// TwinCAT 3 PLC project IvS_Alpaca
// ProgramVersion: 3.1.4024.0
// libraries:
//   Tc2_Standard, * (Beckhoff Automation GmbH)
//   Tc2_System, * (Beckhoff Automation GmbH)
//   Tc2_Utilities, * (Beckhoff Automation GmbH)
//   Tc3_IotBase, * (Beckhoff Automation GmbH)
//   Tc3_JsonXml, * (Beckhoff Automation GmbH)
//   Tc3_Module, * (Beckhoff Automation GmbH)
//   VisuDialogs, * (System)
// project tree:
//   DUTs/Alpaca/ E_AlpacaCoverState.TcDUT, E_AlpacaStatusCode.TcDUT, ST_AlpacaGetBool.TcDUT, ST_AlpacaGetCoverState.TcDUT, ST_AlpacaGetDint.TcDUT, ST_AlpacaGetLreal.TcDUT, ST_AlpacaGetRequest.TcDUT, ST_AlpacaPutMove.TcDUT, ST_AlpacaPutNoArgs.TcDUT, ST_AlpacaPutRequest.TcDUT, ST_AlpacaPutSlewToAltAz.TcDUT, ST_AlpacaPutSlewToCoordinates.TcDUT, ST_AlpacaPutTracking.TcDUT
//   DUTs/AsaTelescope/ E_AsaTelescopeRequests.TcDUT, ST_AsaTelescopeGetters.TcDUT, ST_AsaTelescopePutters.TcDUT
//   / GlobalTextList.TcGTLO, PlcTask.TcTTO, Visualization Manager.TcVMO (not stored)
//   POUs/Alpaca/ FB_AlpacaGet.TcPOU, FB_AlpacaPut.TcPOU, F_AlpacaFormatUri.TcPOU
//   POUs/AsaTelescope/ FB_AsaTelescope.TcPOU
//   POUs/ MAIN.TcPOU
//   VISUs/Alpaca/ VISU_AlpacaGetBool.TcVIS, VISU_AlpacaGetCoverState.TcVIS, VISU_AlpacaGetLreal.TcVIS, VISU_AlpacaPutMove.TcVIS, VISU_AlpacaPutNoArgs.TcVIS, VISU_AlpacaPutRequest.TcVIS, VISU_AlpacaPutSlewToAltAz.TcVIS, VISU_AlpacaPutSlewToCoordinates.TcVIS, VISU_AlpacaPutTracking.TcVIS
//   VISUs/AsaTelescope/ VISU_AsaTelescope.TcVIS
//   VISUs/ VISU_MAIN.TcVIS
// real-time tasks:
//   TASK PlcTask: cycle T#10ms, priority 20, ADS port 350

CONFIGURATION IvS_Alpaca
    RESOURCE PLC ON TwinCAT3
        TASK PlcTask(INTERVAL := T#10ms, PRIORITY := 20);
        PROGRAM MAIN WITH PlcTask : MAIN;
    END_RESOURCE
END_CONFIGURATION

// ---- DUTs/Alpaca/E_AlpacaCoverState.TcDUT
{attribute 'qualified_only'}
{attribute 'to_string'}
TYPE E_AlpacaCoverState :
(
	NOT_PRESENT := 0,
    CLOSED      := 1,
    MOVING      := 2,
    OPEN        := 3,
    UNKNOWN     := 4,
    ERROR       := 5
) DINT := UNKNOWN;
END_TYPE

// ---- DUTs/Alpaca/E_AlpacaStatusCode.TcDUT
{attribute 'qualified_only'}
{attribute 'strict'}
TYPE E_AlpacaStatusCode :
(
    NOTSET                          := 0,
	OK                              := 1,
    ERROR                           := 2,
    ERROR_WRONG_CONVERSION          := 3,
    ERROR_WRONG_RESPONSE_MEMBER     := 4,
    ERROR_WRONG_RESPONSE_CONTENT    := 5,
    ERROR_WRONG_HTTP_STATUS_CODE    := 6,
    ERROR_OTHER_COMMAND_SCHEDULED   := 7
);
END_TYPE

// ---- DUTs/Alpaca/ST_AlpacaGetBool.TcDUT
TYPE ST_AlpacaGetBool EXTENDS ST_AlpacaGetRequest:
STRUCT
    bValue : BOOL;
END_STRUCT
END_TYPE

// ---- DUTs/Alpaca/ST_AlpacaGetCoverState.TcDUT
TYPE ST_AlpacaGetCoverState EXTENDS ST_AlpacaGetDint :
STRUCT
    eValue : E_AlpacaCoverState;
    sValue : STRING;
END_STRUCT
END_TYPE

// ---- DUTs/Alpaca/ST_AlpacaGetDint.TcDUT
TYPE ST_AlpacaGetDint EXTENDS ST_AlpacaGetRequest:
STRUCT
    nValue : DINT;
END_STRUCT
END_TYPE

// ---- DUTs/Alpaca/ST_AlpacaGetLreal.TcDUT
TYPE ST_AlpacaGetLreal EXTENDS ST_AlpacaGetRequest:
STRUCT
    lrValue : LREAL;
END_STRUCT
END_TYPE

// ---- DUTs/Alpaca/ST_AlpacaGetRequest.TcDUT
// Common base class for the "Get" requests
TYPE ST_AlpacaGetRequest :
STRUCT
    sName       : STRING;
    eStatusCode : E_AlpacaStatusCode;
    rAge        : REAL;                 // age of the last reading, in seconds, since the last loop start
END_STRUCT
END_TYPE

// ---- DUTs/Alpaca/ST_AlpacaPutMove.TcDUT
TYPE ST_AlpacaPutMove EXTENDS ST_AlpacaPutRequest:
STRUCT
    // inputs
    i_Position : DINT;
END_STRUCT
END_TYPE

// ---- DUTs/Alpaca/ST_AlpacaPutNoArgs.TcDUT
TYPE ST_AlpacaPutNoArgs EXTENDS ST_AlpacaPutRequest:
STRUCT
    // just for the sake of semantics, our 'No args' structure extends
    // our common "put" request structure, but it doesn't add any members.
END_STRUCT
END_TYPE

// ---- DUTs/Alpaca/ST_AlpacaPutRequest.TcDUT
// Common base class for the "Put" requests
TYPE ST_AlpacaPutRequest :
STRUCT
    sName           : STRING;
    bExecute        : BOOL;
    eStatusCode     : E_AlpacaStatusCode;
    nErrorCode      : DINT;
    sErrorMessage   : STRING;
END_STRUCT
END_TYPE

// ---- DUTs/Alpaca/ST_AlpacaPutSlewToAltAz.TcDUT
TYPE ST_AlpacaPutSlewToAltAz EXTENDS ST_AlpacaPutRequest:
STRUCT
    // inputs
    i_lrAltitude    : LREAL;
    i_lrAzimuth     : LREAL;
END_STRUCT
END_TYPE

// ---- DUTs/Alpaca/ST_AlpacaPutSlewToCoordinates.TcDUT
TYPE ST_AlpacaPutSlewToCoordinates EXTENDS ST_AlpacaPutRequest:
STRUCT
    // inputs
    i_lrRightAscension  : LREAL;
    i_lrDeclination     : LREAL;
END_STRUCT
END_TYPE

// ---- DUTs/Alpaca/ST_AlpacaPutTracking.TcDUT
TYPE ST_AlpacaPutTracking EXTENDS ST_AlpacaPutRequest:
STRUCT
    // inputs
    i_bTracking : BOOL;
END_STRUCT
END_TYPE

// ---- DUTs/AsaTelescope/E_AsaTelescopeRequests.TcDUT
{attribute 'qualified_only'}
TYPE E_AsaTelescopeRequests :
(
    // the data below gets read continuously in order from top to bottom
    RIGHT_ASCENSION := 0,
    DECLINATION,
    AZIMUTH,
    ALTITUDE,
    SLEWING,
    TARGET_RIGHT_ASCENSION,
    TARGET_DECLINATION,
    M2_POSITION,
    COVER_STATE,
    
    // COMMANDS
    // ==================================================================
    // special state meaning no state requested
    NO_COMMAND,
    // add all commands below (order is not relevant)
    ABORT_SLEW,
    SLEW_TO_ALTAZ,
    SLEW_TO_COORDINATES,
    OPEN_COVER,
    CLOSE_COVER,
    TRACKING,
    M2_MOVE
);
END_TYPE

// ---- DUTs/AsaTelescope/ST_AsaTelescopeGetters.TcDUT
TYPE ST_AsaTelescopeGetters :
STRUCT
    stRightAscension          : ST_AlpacaGetLreal      := (sName := 'Right Ascension');
    stDeclination             : ST_AlpacaGetLreal      := (sName := 'Declination');
    stAzimuth                 : ST_AlpacaGetLreal      := (sName := 'Azimuth');
    stAltitude                : ST_AlpacaGetLreal      := (sName := 'Altitude');
    stSlewing                 : ST_AlpacaGetBool       := (sName := 'Slewing');
    stTargetRightAscension    : ST_AlpacaGetLreal      := (sName := 'Target Right Ascension');
    stTargetDeclination       : ST_AlpacaGetLreal      := (sName := 'Target Declination');
    stM2Position              : ST_AlpacaGetLreal      := (sName := 'M2 position');
    stCoverState              : ST_AlpacaGetCoverState := (sName := 'Cover state');
END_STRUCT
END_TYPE

// ---- DUTs/AsaTelescope/ST_AsaTelescopePutters.TcDUT
TYPE ST_AsaTelescopePutters :
STRUCT
    stAbortSlew   : ST_AlpacaPutNoArgs              := (sName := 'Abort slew');
    stSlewToAltAz : ST_AlpacaPutSlewToAltAz         := (sName := 'Slew to Alt Az');
    stSlewToCoo   : ST_AlpacaPutSlewToCoordinates   := (sName := 'Slew to coordinates');
    stOpenCover   : ST_AlpacaPutNoArgs              := (sName := 'Open cover');
    stCloseCover  : ST_AlpacaPutNoArgs              := (sName := 'Close cover');
    stTracking    : ST_AlpacaPutTracking            := (sName := 'Tracking');
    stM2Move      : ST_AlpacaPutMove                := (sName := 'M2 move');
END_STRUCT
END_TYPE

// ---- POUs/MAIN.TcPOU
PROGRAM MAIN
VAR
    {attribute 'OPC.UA.DA':='1'}
    fbTelescope : FB_AsaTelescope( 
          // sTelHost := '10.33.179.130', nTelPort := 11111, sAccHost := 'localhost', nAccPort := 11112); // Leuven
             sTelHost := 'localhost', nTelPort := 32323, sAccHost := 'localhost', nAccPort := 32323); // Simulator
END_VAR

fbTelescope();

END_PROGRAM

// ---- POUs/AsaTelescope/FB_AsaTelescope.TcPOU
FUNCTION_BLOCK FB_AsaTelescope
VAR_INPUT
    {attribute 'OPC.UA.DA':='0'}
    sTelHost            : STRING;           // Telescope hostname or IP address
    {attribute 'OPC.UA.DA':='0'}
    nTelPort            : UINT;             // Telescope port
    {attribute 'OPC.UA.DA':='0'}
    sAccHost            : STRING;           // Accessory hostname or IP address
    {attribute 'OPC.UA.DA':='0'}
    nAccPort            : UINT;             // Accessory port
    {attribute 'OPC.UA.DA':='0'}
    nLoopTime           : UINT   := 1000;   // Minimum loop time in ms (so we will wait if the loop is finished earlier)
END_VAR
VAR_OUTPUT
    {attribute 'OPC.UA.DA' := '1'}
    stData              : ST_AsaTelescopeGetters;
    {attribute 'OPC.UA.DA' := '1'}
    stCommands          : ST_AsaTelescopePutters;
    {attribute 'OPC.UA.DA' := '1'}
    bTelConnected       : BOOL;
    {attribute 'OPC.UA.DA' := '1'}
    bAccConnected       : BOOL;
END_VAR
VAR
    // store the HTTP client parameters that are really used
    {attribute 'OPC.UA.DA':='0'}
    sTrueTelHost        : STRING;
    {attribute 'OPC.UA.DA':='0'}
    sTrueAccHost        : STRING;
    {attribute 'OPC.UA.DA':='0'}
    nTrueTelPort        : UINT;
    {attribute 'OPC.UA.DA':='0'}
    nTrueAccPort        : UINT;
    {attribute 'OPC.UA.DA':='0'}
    bResetTel           : BOOL;
    {attribute 'OPC.UA.DA':='0'}
    bResetAcc           : BOOL;

    // keep track of the current state and the next state
    // - getters (fbGet...) will be read in order of E_AlpacaRequest
    // - putters (fbPut...) can be "scheduled" by setting eNextState to the requested command.
    //   As soon as the current request is finished, the CASE OF will therefore jump
    //   to the new command
    {attribute 'OPC.UA.DA':='0'}
    eState              : E_AsaTelescopeRequests;
    {attribute 'OPC.UA.DA':='0'}
    eNextState          : E_AsaTelescopeRequests := E_AsaTelescopeRequests.NO_COMMAND;
    
    // create the 2 necessary clients for the telescope
    {attribute 'OPC.UA.DA':='0'}
    fbClientTel         : FB_IotHttpClient;
    {attribute 'OPC.UA.DA':='0'}
    fbClientAcc         : FB_IotHttpClient;
    
    // data (read)
    {attribute 'OPC.UA.DA':='0'}
    fbGetTelRA          : FB_AlpacaGet('telescope', 0, 'rightascension');
    {attribute 'OPC.UA.DA':='0'}
    fbGetTelDec         : FB_AlpacaGet('telescope', 0, 'declination');
    {attribute 'OPC.UA.DA':='0'}
    fbGetTelAz          : FB_AlpacaGet('telescope', 0, 'azimuth');
    {attribute 'OPC.UA.DA':='0'}
    fbGetTelAlt         : FB_AlpacaGet('telescope', 0, 'altitude');
    {attribute 'OPC.UA.DA':='0'}
    fbGetTelSlew        : FB_AlpacaGet('telescope', 0, 'slewing');
    {attribute 'OPC.UA.DA':='0'}
    fbGetTelTRA         : FB_AlpacaGet('telescope', 0, 'targetrightascension');
    {attribute 'OPC.UA.DA':='0'}
    fbGetTelTDec        : FB_AlpacaGet('telescope', 0, 'targetdeclination');
    {attribute 'OPC.UA.DA':='0'}
    fbGetFocPos         : FB_AlpacaGet('focuser', 0, 'position');
    {attribute 'OPC.UA.DA':='0'}
    fbGetCovState       : FB_AlpacaGet('covercalibrator', 0, 'coverstate');
    
    // commands (write)
    {attribute 'OPC.UA.DA':='0'}
    fbPutTelAbortSlew   : FB_AlpacaPut('telescope', 0, 'abortslew');
    {attribute 'OPC.UA.DA':='0'}
    fbPutTelSlewAltAz   : FB_AlpacaPut('telescope', 0, 'slewtoaltazasync');
    {attribute 'OPC.UA.DA':='0'}
    fbPutTelSlewCoo     : FB_AlpacaPut('telescope', 0, 'slewtocoordinatesasync');
    {attribute 'OPC.UA.DA':='0'}
    fbPutCovOpen        : FB_AlpacaPut('covercalibrator', 0, 'opencover');
    {attribute 'OPC.UA.DA':='0'}
    fbPutCovClose       : FB_AlpacaPut('covercalibrator', 0, 'closecover');
    {attribute 'OPC.UA.DA':='0'}
    fbPutTelTracking    : FB_AlpacaPut('telescope', 0, 'tracking');
    {attribute 'OPC.UA.DA':='0'}
    fbPutFocMove        : FB_AlpacaPut('focuser', 0, 'move');
    
    // cycle time variables
    {attribute 'OPC.UA.DA':='0'}
    tStart              : TIME;
END_VAR

IF sTrueTelHost <> sTelHost OR nTrueTelPort <> nTelPort THEN
    bResetTel := TRUE;
END_IF
IF sTrueAccHost <> sAccHost OR nTrueAccPort <> nAccPort THEN
    bResetAcc := TRUE;
END_IF

IF bResetTel THEN
    fbClientTel.Disconnect();
    sTrueTelHost := sTelHost;
    nTrueTelPort := nTelPort;
    
    IF NOT fbClientTel.bConfigured THEN 	
        fbClientTel.sHostName := sTrueTelHost;
        fbClientTel.nHostPort := nTrueTelPort;
        fbClientTel.bKeepAlive := TRUE;
        fbClientTel.tConnectionTimeout := T#3s;
        fbClientTel.stTLS.bNoServerCertCheck := FALSE;
        bResetTel := FALSE;
        fbClientTel.Execute();
    END_IF
ELSE
    fbClientTel.Execute();
END_IF


IF bResetAcc THEN
    fbClientAcc.Disconnect();
    sTrueAccHost := sAccHost;
    nTrueAccPort := nAccPort;
    
    IF NOT fbClientAcc.bConfigured THEN 	
        fbClientAcc.sHostName := sTrueAccHost;
        fbClientAcc.nHostPort := nTrueAccPort;
        fbClientAcc.bKeepAlive := TRUE;
        fbClientAcc.tConnectionTimeout := T#3s;
        fbClientAcc.stTLS.bNoServerCertCheck := FALSE;
        bResetAcc := FALSE;
        fbClientAcc.Execute();
    END_IF
ELSE
    fbClientAcc.Execute();
END_IF

bTelConnected := fbClientTel.bConnected;
bAccConnected := fbClientAcc.bConnected;

eNextState := M_GetNextCommand();

CASE eState OF
    E_AsaTelescopeRequests.RIGHT_ASCENSION:
        tStart := TIME();
        M_ReadLreal(fbClientTel, fbGetTelRA   , stData.stRightAscension);
    E_AsaTelescopeRequests.DECLINATION:
        M_ReadLreal(fbClientTel, fbGetTelDec  , stData.stDeclination);
    E_AsaTelescopeRequests.AZIMUTH:
        M_ReadLreal(fbClientTel, fbGetTelAz   , stData.stAzimuth);
    E_AsaTelescopeRequests.ALTITUDE:
        M_ReadLreal(fbClientTel, fbGetTelAlt  , stData.stAltitude);
    E_AsaTelescopeRequests.SLEWING:
        M_ReadBool(fbClientTel, fbGetTelSlew  , stData.stSlewing);
    E_AsaTelescopeRequests.TARGET_RIGHT_ASCENSION:
        M_ReadLreal(fbClientTel, fbGetTelTRA  , stData.stTargetRightAscension);
    E_AsaTelescopeRequests.TARGET_DECLINATION:
        M_ReadLreal(fbClientTel, fbGetTelTDec , stData.stTargetDeclination);
    E_AsaTelescopeRequests.M2_POSITION:
        M_ReadLreal(fbClientAcc, fbGetFocPos , stData.stM2Position);
    E_AsaTelescopeRequests.COVER_STATE:
        M_ReadCoverState(fbClientAcc, fbGetCovState , stData.stCoverState);
    // Special state, used to wait for the next loop
    E_AsaTelescopeRequests.NO_COMMAND:
        M_UpdateState();
    // Commands
    E_AsaTelescopeRequests.ABORT_SLEW:
        M_WriteNoArgs(fbClientTel, fbPutTelAbortSlew , stCommands.stAbortSlew);
    E_AsaTelescopeRequests.SLEW_TO_ALTAZ:
        M_WriteSlewToAltAz(fbClientTel, fbPutTelSlewAltAz , stCommands.stSlewToAltAz);
    E_AsaTelescopeRequests.SLEW_TO_COORDINATES:
        M_WriteSlewToCoordinates(fbClientTel, fbPutTelSlewCoo , stCommands.stSlewToCoo);
    E_AsaTelescopeRequests.OPEN_COVER:
        M_WriteNoArgs(fbClientAcc, fbPutCovOpen , stCommands.stOpenCover);
    E_AsaTelescopeRequests.CLOSE_COVER:
        M_WriteNoArgs(fbClientAcc, fbPutCovClose , stCommands.stCloseCover);
    E_AsaTelescopeRequests.TRACKING:
        M_WriteTracking(fbClientTel, fbPutTelTracking , stCommands.stTracking);
    E_AsaTelescopeRequests.M2_MOVE:
        M_WriteMove(fbClientAcc, fbPutFocMove , stCommands.stM2Move);
    ELSE
        // this should never happen, but to be sure let's restart
        eState := E_AsaTelescopeRequests.RIGHT_ASCENSION;
END_CASE

METHOD FB_init : BOOL
VAR_INPUT
	bInitRetains : BOOL; // if TRUE, the retain variables are initialized (warm start / cold start)
	bInCopyCode : BOOL;  // if TRUE, the instance afterwards gets moved into the copy code (online change)
    sTelHost            : STRING    := 'localhost'; // Telescope hostname or IP address
    nTelPort            : UINT      := 11111;       // Telescope port
    sAccHost            : STRING    := 'localhost'; // Accessory hostname or IP address
    nAccPort            : UINT      := 11112;       // Accessory port
END_VAR
THIS^.sTelHost := sTelHost;
THIS^.nTelPort := nTelPort;
THIS^.sAccHost := sAccHost;
THIS^.nAccPort := nAccPort;
END_METHOD

METHOD M_GetAge : REAL
VAR_INPUT
END_VAR
M_GetAge := TIME_TO_REAL(TIME() - tStart) / 1000.0;
END_METHOD

METHOD M_GetNextCommand : E_AsaTelescopeRequests
VAR_INPUT
END_VAR
IF stCommands.stAbortSlew.bExecute THEN
    M_GetNextCommand := E_AsaTelescopeRequests.ABORT_SLEW;
ELSIF stCommands.stCloseCover.bExecute THEN
    M_GetNextCommand := E_AsaTelescopeRequests.CLOSE_COVER;
ELSIF stCommands.stOpenCover.bExecute THEN
    M_GetNextCommand := E_AsaTelescopeRequests.OPEN_COVER;
ELSIF stCommands.stSlewToAltAz.bExecute THEN
    M_GetNextCommand := E_AsaTelescopeRequests.SLEW_TO_ALTAZ;
ELSIF stCommands.stSlewToCoo.bExecute THEN
    M_GetNextCommand := E_AsaTelescopeRequests.SLEW_TO_COORDINATES;
ELSIF stCommands.stTracking.bExecute THEN
    M_GetNextCommand := E_AsaTelescopeRequests.TRACKING;
ELSIF stCommands.stM2Move.bExecute THEN
    M_GetNextCommand := E_AsaTelescopeRequests.M2_MOVE;
ELSE
    M_GetNextCommand := E_AsaTelescopeRequests.NO_COMMAND;
END_IF
END_METHOD

METHOD M_ReadBool : BOOL
VAR_INPUT
END_VAR
VAR_IN_OUT
    fbClient : FB_IotHttpClient;
    fbRequest : FB_AlpacaGet;
    Data : ST_AlpacaGetBool;
END_VAR
fbRequest(fbClient := fbClient); 

IF NOT fbRequest.bBusy THEN
    IF fbRequest.bError THEN
        // let's update only the statuscode, and leave the rest as is
        Data.eStatusCode := E_AlpacaStatusCode.ERROR; 
    ELSE
        fbRequest.M_FetchResultBool(Data);
	END_IF
    Data.rAge := M_GetAge();
    M_UpdateState();
END_IF
END_METHOD

METHOD M_ReadCoverState : BOOL
VAR_INPUT
END_VAR
VAR_IN_OUT
    fbClient : FB_IotHttpClient;
    fbRequest : FB_AlpacaGet;
    Data : ST_AlpacaGetCoverState;
END_VAR
fbRequest(fbClient := fbClient); 

IF NOT fbRequest.bBusy THEN
    IF fbRequest.bError THEN
        // let's update only the statuscode, and leave the rest as is
        Data.eStatusCode := E_AlpacaStatusCode.ERROR; 
    ELSE
        fbRequest.M_FetchResultCoverState(Data);
	END_IF
    Data.rAge := M_GetAge();
    M_UpdateState();
END_IF
END_METHOD

METHOD M_ReadLreal : BOOL
VAR_INPUT
END_VAR
VAR_IN_OUT
    fbClient : FB_IotHttpClient;
    fbRequest : FB_AlpacaGet;
    Data : ST_AlpacaGetLreal;
END_VAR
fbRequest(fbClient := fbClient); 

IF NOT fbRequest.bBusy THEN
    IF fbRequest.bError THEN
        // let's update only the statuscode, and leave the rest as is
        Data.eStatusCode := E_AlpacaStatusCode.ERROR; 
    ELSE
        fbRequest.M_FetchResultLreal(Data);
	END_IF
    Data.rAge := M_GetAge();
    M_UpdateState();
END_IF
END_METHOD

METHOD M_ScheduleRpcCall : E_AlpacaStatusCode
VAR_INPUT
    eCheck : E_AsaTelescopeRequests; 
END_VAR
VAR_IN_OUT
    tPut : ST_AlpacaPutRequest; 
END_VAR
tPut.bExecute := TRUE;

// check if our command is really scheduled
// (which means: check if no other command was scheduled instead)
IF M_GetNextCommand() = eCheck THEN
    M_ScheduleRpcCall := E_AlpacaStatusCode.OK;
ELSE
    M_ScheduleRpcCall := E_AlpacaStatusCode.ERROR_OTHER_COMMAND_SCHEDULED;
END_IF
END_METHOD

METHOD M_UpdateState : BOOL
VAR_INPUT
END_VAR
IF eNextState > E_AsaTelescopeRequests.NO_COMMAND THEN
    // command scheduled!
    eState := eNextState;
    eNextState := E_AsaTelescopeRequests.NO_COMMAND;
ELSE
    IF eState = E_AsaTelescopeRequests.NO_COMMAND THEN
        IF TIME() > tStart + UINT_TO_TIME(nLoopTime) THEN
            eState := 0;
        END_IF 
	ELSIF eState < E_AsaTelescopeRequests.NO_COMMAND THEN
        eState := eState + 1;
    ELSE
        eState := 0;
    END_IF
END_IF
END_METHOD

METHOD M_WriteMove : BOOL
VAR_INPUT
END_VAR
VAR_IN_OUT
    fbClient    : FB_IotHttpClient;
    fbPut       : FB_AlpacaPut;
    tRequest    : ST_AlpacaPutMove;
END_VAR
IF NOT fbPut.bBusy THEN
    fbPut.sArguments := CONCAT('Position=', DINT_TO_STRING(tRequest.i_Position));
END_IF

fbPut(fbClient := fbClient); 

IF NOT fbPut.bBusy THEN
    IF fbPut.bError THEN
        // let's update only the statuscode, and leave the rest as is
        tRequest.eStatusCode := E_AlpacaStatusCode.ERROR; 
    ELSE
        fbPut.M_FetchResult(tRequest);
	END_IF
    tRequest.bExecute := FALSE;
    M_UpdateState();
END_IF
END_METHOD

METHOD M_WriteNoArgs : BOOL
VAR_INPUT
END_VAR
VAR_IN_OUT
    fbClient    : FB_IotHttpClient;
    fbPut       : FB_AlpacaPut;
    tRequest    : ST_AlpacaPutRequest;
END_VAR
fbPut(fbClient := fbClient); 

IF NOT fbPut.bBusy THEN
    IF fbPut.bError THEN
        // let's update only the statuscode, and leave the rest as is
        tRequest.eStatusCode := E_AlpacaStatusCode.ERROR; 
    ELSE
        fbPut.M_FetchResult(tRequest);
	END_IF
    tRequest.bExecute := FALSE;
    M_UpdateState();
END_IF
END_METHOD

METHOD M_WriteSlewToAltAz : BOOL
VAR_INPUT
END_VAR
VAR_IN_OUT
    fbClient    : FB_IotHttpClient;
    fbPut       : FB_AlpacaPut;
    tRequest    : ST_AlpacaPutSlewToAltAz;
END_VAR
IF NOT fbPut.bBusy THEN
    fbPut.sArguments := CONCAT('Azimuth=',
                       CONCAT(LREAL_TO_STRING(tRequest.i_lrAzimuth),
                       CONCAT('&Altitude=', 
                              LREAL_TO_STRING(tRequest.i_lrAltitude))));
END_IF

fbPut(fbClient := fbClient); 

IF NOT fbPut.bBusy THEN
    IF fbPut.bError THEN
        // let's update only the statuscode, and leave the rest as is
        tRequest.eStatusCode := E_AlpacaStatusCode.ERROR; 
    ELSE
        fbPut.M_FetchResult(tRequest);
	END_IF
    tRequest.bExecute := FALSE;
    M_UpdateState();
END_IF
END_METHOD

METHOD M_WriteSlewToCoordinates : BOOL
VAR_INPUT
END_VAR
VAR_IN_OUT
    fbClient    : FB_IotHttpClient;
    fbPut       : FB_AlpacaPut;
    tRequest    : ST_AlpacaPutSlewToCoordinates;
END_VAR
IF NOT fbPut.bBusy THEN
    fbPut.sArguments := CONCAT('RightAscension=',
                       CONCAT(LREAL_TO_STRING(tRequest.i_lrRightAscension),
                       CONCAT('&Declination=', 
                              LREAL_TO_STRING(tRequest.i_lrDeclination))));
END_IF

fbPut(fbClient := fbClient); 

IF NOT fbPut.bBusy THEN
    IF fbPut.bError THEN
        // let's update only the statuscode, and leave the rest as is
        tRequest.eStatusCode := E_AlpacaStatusCode.ERROR; 
    ELSE
        fbPut.M_FetchResult(tRequest);
	END_IF
    tRequest.bExecute := FALSE;
    M_UpdateState();
END_IF
END_METHOD

METHOD M_WriteTracking : BOOL
VAR_INPUT
END_VAR
VAR_IN_OUT
    fbClient    : FB_IotHttpClient;
    fbPut       : FB_AlpacaPut;
    tRequest    : ST_AlpacaPutTracking;
END_VAR
IF NOT fbPut.bBusy THEN
    IF tRequest.i_bTracking THEN
        fbPut.sArguments := 'Tracking=true';
    ELSE
        fbPut.sArguments := 'Tracking=false';
	END_IF
END_IF

fbPut(fbClient := fbClient); 

IF NOT fbPut.bBusy THEN
    IF fbPut.bError THEN
        // let's update only the statuscode, and leave the rest as is
        tRequest.eStatusCode := E_AlpacaStatusCode.ERROR; 
    ELSE
        fbPut.M_FetchResult(tRequest);
	END_IF
    tRequest.bExecute := FALSE;
    M_UpdateState();
END_IF
END_METHOD

{attribute 'TcRpcEnable':='1'}
METHOD RPC_AbortSlew : E_AlpacaStatusCode
VAR_INPUT
END_VAR
RPC_AbortSlew := M_ScheduleRpcCall(
    tPut    := stCommands.stAbortSlew, 
    eCheck  := E_AsaTelescopeRequests.ABORT_SLEW);
END_METHOD

{attribute 'TcRpcEnable':='1'}
METHOD RPC_CloseCover : E_AlpacaStatusCode
VAR_INPUT
END_VAR
RPC_CloseCover := M_ScheduleRpcCall(
    tPut    := stCommands.stCloseCover, 
    eCheck  := E_AsaTelescopeRequests.CLOSE_COVER);
END_METHOD

{attribute 'TcRpcEnable':='1'}
METHOD RPC_M2Move : E_AlpacaStatusCode
VAR_INPUT
END_VAR
RPC_M2Move := M_ScheduleRpcCall(
    tPut    := stCommands.stM2Move, 
    eCheck  := E_AsaTelescopeRequests.M2_MOVE);
END_METHOD

{attribute 'TcRpcEnable':='1'}
METHOD RPC_OpenCover : E_AlpacaStatusCode
VAR_INPUT
END_VAR
RPC_OpenCover := M_ScheduleRpcCall(
    tPut    := stCommands.stOpenCover, 
    eCheck  := E_AsaTelescopeRequests.OPEN_COVER);
END_METHOD

{attribute 'TcRpcEnable':='1'}
METHOD RPC_SlewToAltAz : E_AlpacaStatusCode
VAR_INPUT
    lrAltitude : LREAL;
    lrAzimuth : LREAL;
END_VAR
stCommands.stSlewToAltAz.i_lrAltitude := lrAltitude;
stCommands.stSlewToAltAz.i_lrAzimuth  := lrAzimuth;

RPC_SlewToAltAz := M_ScheduleRpcCall(
    tPut    := stCommands.stSlewToAltAz, 
    eCheck  := E_AsaTelescopeRequests.SLEW_TO_ALTAZ);
END_METHOD

{attribute 'TcRpcEnable':='1'}
METHOD RPC_SlewToCoordinates : E_AlpacaStatusCode
VAR_INPUT
    lrRightAscension : LREAL;
    lrDeclination : LREAL;
END_VAR
stCommands.stSlewToCoo.i_lrRightAscension    := lrRightAscension;
stCommands.stSlewToCoo.i_lrDeclination       := lrDeclination;

RPC_SlewToCoordinates := M_ScheduleRpcCall(
    tPut    := stCommands.stSlewToCoo, 
    eCheck  := E_AsaTelescopeRequests.SLEW_TO_COORDINATES);
END_METHOD

{attribute 'TcRpcEnable':='1'}
METHOD RPC_Tracking : E_AlpacaStatusCode
VAR_INPUT
    bTracking : BOOL;
END_VAR
stCommands.stTracking.i_bTracking := bTracking;

RPC_Tracking := M_ScheduleRpcCall(
    tPut    := stCommands.stTracking, 
    eCheck  := E_AsaTelescopeRequests.TRACKING);
END_METHOD

END_FUNCTION_BLOCK

// ---- POUs/Alpaca/FB_AlpacaGet.TcPOU
FUNCTION_BLOCK FB_AlpacaGet
VAR_INPUT
END_VAR
VAR_OUTPUT
	bBusy               : BOOL;
	bError              : BOOL;
    eStatusCode         : E_AlpacaStatusCode;
END_VAR
VAR_IN_OUT
    fbClient            : FB_IotHttpClient;
END_VAR
VAR
    sUri                : STRING;
    fbRequest           : FB_IotHttpRequest;
	fbJson              : FB_JsonDomParser;
    nState              : UINT;
	jsonDoc             : SJsonValue;
    jsonVal             : SJsonValue;
	bGetContentResult	: BOOL;
	sContent			: STRING(511);
    tSent               : TIME;
END_VAR

// small state machine:
CASE nState OF 
    0:
        // send the request
        IF fbRequest.SendRequest(
                sUri            := sUri,
                fbClient        := fbClient,
                eRequestType    := ETcIotHttpRequestType.HTTP_GET,
                pContent        := 0,
                nContentSize    := 0, 
                fbHeader        := 0) THEN
            nState      := 1;
            bBusy       := TRUE;
            bError      := FALSE;
            eStatusCode := E_AlpacaStatusCode.OK; 
            tSent       := TIME();
        END_IF
    1:
        // wait for the response
        IF NOT fbRequest.bBusy THEN
            bGetContentResult:= fbRequest.GetContent(
                pContent            := ADR(sContent),
                nContentSize        := SIZEOF(sContent),
                bSetNullTermination := TRUE);
            
			IF fbRequest.nStatusCode >= 200 AND fbRequest.nStatusCode < 300 THEN
				jsonDoc := fbRequest.GetJsonDomContent(fbJson);
				IF jsonDoc <> 0 THEN
                    eStatusCode := E_AlpacaStatusCode.OK; 
					bError:= FALSE;
                ELSE
                    bError := TRUE;
                    eStatusCode := E_AlpacaStatusCode.ERROR_WRONG_RESPONSE_CONTENT; 
				END_IF
            ELSE
                bError := TRUE;
                eStatusCode := E_AlpacaStatusCode.ERROR_WRONG_HTTP_STATUS_CODE; 
			END_IF
                
            nState:= 0;
		    bBusy:= FALSE;
		END_IF
END_CASE

METHOD FB_init : BOOL
VAR_INPUT
	bInitRetains : BOOL; // if TRUE, the retain variables are initialized (warm start / cold start)
	bInCopyCode : BOOL;  // if TRUE, the instance afterwards gets moved into the copy code (online change)
    sDeviceName     : STRING;
    nDeviceNumber   : UINT;
    sVariableName   : STRING;
END_VAR
sUri := F_AlpacaFormatUri(sDeviceName, nDeviceNumber, sVariableName);
END_METHOD

METHOD M_FetchResultBool : BOOL
VAR_INPUT
END_VAR
VAR_IN_OUT
    stData : ST_AlpacaGetBool;
END_VAR
VAR
    nTmpInt : DINT;
END_VAR
IF fbJson.HasMember(jsonDoc, 'Value') THEN
    jsonVal:= fbJson.FindMember(jsonDoc, 'Value');
    IF fbJson.IsBool(jsonVal) THEN
        stData.bValue      := fbJson.GetBool(jsonVal);
        stData.eStatusCode := E_AlpacaStatusCode.OK;
        stData.rAge       := TIME_TO_REAL(TIME() - tSent);
    ELSIF fbJson.IsInt(jsonVal) THEN
        nTmpInt := fbJson.GetInt(jsonVal);
        IF nTmpInt = 0 THEN
            stData.bValue := FALSE;
            stData.eStatusCode := E_AlpacaStatusCode.OK;
            stData.rAge       := TIME_TO_REAL(TIME() - tSent);
        ELSIF nTmpInt = 1 THEN
            stData.bValue := TRUE;
            stData.eStatusCode := E_AlpacaStatusCode.OK;
            stData.rAge       := TIME_TO_REAL(TIME() - tSent);
        ELSE
            stData.bValue      := FALSE;
            stData.eStatusCode := E_AlpacaStatusCode.ERROR_WRONG_CONVERSION;
		END_IF
    ELSE
        stData.bValue      := FALSE;
        stData.eStatusCode := E_AlpacaStatusCode.ERROR_WRONG_CONVERSION;
	END_IF
ELSE
    stData.bValue      := FALSE;
    stData.eStatusCode := E_AlpacaStatusCode.ERROR_WRONG_RESPONSE_MEMBER;
END_IF
END_METHOD

METHOD M_FetchResultCoverState : BOOL
VAR_INPUT
END_VAR
VAR_IN_OUT
    stData : ST_AlpacaGetCoverState;
END_VAR
VAR
    nTmpInt : DINT;
END_VAR
IF fbJson.HasMember(jsonDoc, 'Value') THEN
    jsonVal:= fbJson.FindMember(jsonDoc, 'Value');
    IF fbJson.IsInt(jsonVal) THEN
        stData.nValue       := fbJson.GetInt(jsonVal);
        stData.eValue       := stData.nValue;
        stData.sValue       := TO_STRING(stData.eValue);
        stData.eStatusCode  := E_AlpacaStatusCode.OK;
        stData.rAge         := TIME_TO_REAL(TIME() - tSent);
    ELSE
        stData.eValue       := E_AlpacaCoverState.UNKNOWN;
        stData.nValue       := stData.eValue;
        stData.sValue       := TO_STRING(stData.eValue);
        stData.eStatusCode  := E_AlpacaStatusCode.ERROR_WRONG_CONVERSION;
	END_IF
ELSE
    stData.eValue       := E_AlpacaCoverState.UNKNOWN;
    stData.nValue       := stData.eValue;
    stData.sValue       := TO_STRING(stData.eValue);
    stData.eStatusCode := E_AlpacaStatusCode.ERROR_WRONG_RESPONSE_MEMBER;
END_IF
END_METHOD

METHOD M_FetchResultLreal : LREAL
VAR_INPUT
END_VAR
VAR_IN_OUT
    stData : ST_AlpacaGetLreal;
END_VAR
IF fbJson.HasMember(jsonDoc, 'Value') THEN
    jsonVal:= fbJson.FindMember(jsonDoc, 'Value');
    IF fbJson.IsDouble(jsonVal) THEN
        stData.lrValue      := fbJson.GetDouble(jsonVal);
        stData.eStatusCode  := E_AlpacaStatusCode.OK;
        stData.rAge         := TIME_TO_REAL(TIME() - tSent);
    ELSIF fbJson.IsInt(jsonVal) THEN
        stData.lrValue      := DINT_TO_LREAL(fbJson.GetInt(jsonVal));
        stData.eStatusCode  := E_AlpacaStatusCode.OK;
        stData.rAge         := TIME_TO_REAL(TIME() - tSent);
    ELSE
        stData.lrValue      := 0.0;
        stData.eStatusCode  := E_AlpacaStatusCode.ERROR_WRONG_CONVERSION;
	END_IF
ELSE
    stData.lrValue          := 0.0;
    stData.eStatusCode      := E_AlpacaStatusCode.ERROR_WRONG_RESPONSE_MEMBER;
END_IF
END_METHOD

END_FUNCTION_BLOCK

// ---- POUs/Alpaca/F_AlpacaFormatUri.TcPOU
FUNCTION F_AlpacaFormatUri : STRING
VAR_INPUT
    sDeviceName     : STRING;
    nDeviceNumber   : UINT;
    sVariableName   : STRING;
END_VAR
VAR
END_VAR

F_AlpacaFormatUri := CONCAT('/api/v1/',
                     CONCAT(sDeviceName,
                     CONCAT('/',
                     CONCAT(UINT_TO_STRING(nDeviceNumber),
                     CONCAT('/', sVariableName)))));

END_FUNCTION

// ---- POUs/Alpaca/FB_AlpacaPut.TcPOU
FUNCTION_BLOCK FB_AlpacaPut
VAR_INPUT
	sArguments			: STRING(511);
END_VAR
VAR_OUTPUT
	bBusy               : BOOL;
	bError              : BOOL;
    eStatusCode         : E_AlpacaStatusCode;
    sResult             : SJsonValue;
END_VAR
VAR_IN_OUT
    fbClient            : FB_IotHttpClient;
END_VAR
VAR
    sUri                : STRING;
	sSend			    : STRING(511);
    fbRequest           : FB_IotHttpRequest;
	fbJson              : FB_JsonDomParser;
    nState              : UINT;
    jsonVal             : SJsonValue;
	bGetContentResult	: BOOL;
	sContent			: STRING(511);
    tSent               : TIME;
END_VAR

fbRequest.sContentType := 'application/x-www-form-urlencoded';

// small state machine:
CASE nState OF 
    0:
        // send the command
        sSend := 'ClientID=1';
        IF LEN2(ADR(sArguments)) > 0 THEN
            sSend := CONCAT(sSend, CONCAT('&', sArguments));
		END_IF
        // send the request
        IF fbRequest.SendRequest(
                sUri            := sUri,
                fbClient        := fbClient,
                eRequestType    := ETcIotHttpRequestType.HTTP_PUT,
                pContent        := ADR(sSend),
                nContentSize    := LEN2(ADR(sSend)), 
                fbHeader        := 0) THEN
            nState := 1;
            bBusy  := TRUE;
            bError := FALSE;
            eStatusCode := E_AlpacaStatusCode.OK; 
            tSent       := TIME();
        END_IF
    1:
        // wait for the response
        IF NOT fbRequest.bBusy THEN
            bGetContentResult:= fbRequest.GetContent(
                pContent            := ADR(sContent),
                nContentSize        := SIZEOF(sContent),
                bSetNullTermination := TRUE);
            
			IF fbRequest.nStatusCode >= 200 AND fbRequest.nStatusCode < 300 THEN
				sResult := fbRequest.GetJsonDomContent(fbJson);
				IF sResult <> 0 THEN
                    eStatusCode := E_AlpacaStatusCode.OK; 
					bError:= FALSE;
                ELSE
                    bError := TRUE;
                    eStatusCode := E_AlpacaStatusCode.ERROR_WRONG_RESPONSE_CONTENT; 
				END_IF
            ELSE
                bError := TRUE;
                eStatusCode := E_AlpacaStatusCode.ERROR_WRONG_HTTP_STATUS_CODE;        
			END_IF
                
            nState:= 0;
		    bBusy:= FALSE;
		END_IF
END_CASE

METHOD FB_init : BOOL
VAR_INPUT
	bInitRetains    : BOOL; // if TRUE, the retain variables are initialized (warm start / cold start)
	bInCopyCode     : BOOL;  // if TRUE, the instance afterwards gets moved into the copy code (online change)
    sDeviceName     : STRING;
    nDeviceNumber   : UINT;
    sVariableName   : STRING;
END_VAR
sUri := F_AlpacaFormatUri(sDeviceName, nDeviceNumber, sVariableName);
END_METHOD

METHOD M_FetchResult : LREAL
VAR_INPUT
END_VAR
VAR_IN_OUT
    stData : ST_AlpacaPutRequest;
END_VAR
IF fbJson.HasMember(sResult, 'ErrorNumber') THEN
    jsonVal:= fbJson.FindMember(sResult, 'ErrorNumber');
    stData.eStatusCode := E_AlpacaStatusCode.OK;
    IF fbJson.IsInt(jsonVal) THEN
        stData.nErrorCode  := fbJson.GetInt(jsonVal);
    ELSE
        stData.eStatusCode := E_AlpacaStatusCode.ERROR_WRONG_CONVERSION;
	END_IF
    
    IF fbJson.HasMember(sResult, 'ErrorMessage') THEN
        jsonVal:= fbJson.FindMember(sResult, 'ErrorMessage');
        IF fbJson.IsString(jsonVal) THEN
            stData.sErrorMessage  := fbJson.GetString(jsonVal);
        ELSE
            stData.eStatusCode := E_AlpacaStatusCode.ERROR_WRONG_CONVERSION;
        END_IF
    END_IF
ELSE
    stData.eStatusCode := E_AlpacaStatusCode.ERROR_WRONG_RESPONSE_MEMBER;
END_IF
END_METHOD

END_FUNCTION_BLOCK

// ---- GlobalTextList.TcGTLO
TEXTLIST GlobalTextList
  313 = '%.2f s'
  43 = '%.3f s'
  604 = '%.6f'
  241 = '%d'
  10 = '%d ms'
  998 = '%s'
  899 = 'ACC host'
  32 = 'ACC port'
  123 = 'Age'
  766 = 'Alt'
  657 = 'Altitude'
  157 = 'Azimuth'
  267 = 'Close cover'
  257 = 'Commands'
  838 = 'Config'
  247 = 'Connected'
  716 = 'Data'
  715 = 'Dec'
  83 = 'Declination'
  780 = 'Error code'
  828 = 'Error message'
  446 = 'Go'
  788 = 'Host name'
  518 = 'IP address'
  555 = 'Loop time'
  204 = 'Loop time [ms]'
  941 = 'Open cover'
  145 = 'Position'
  4 = 'RA'
  436 = 'Result'
  272 = 'Right ascension'
  750 = 'Slew'
  392 = 'Slew to Alt Az'
  983 = 'Slew to Coordinates'
  685 = 'TEL host'
  582 = 'TEL port'
  583 = 'Tracking'
END_TEXTLIST

// ---- VISUs/Alpaca/VISU_AlpacaGetBool.TcVIS
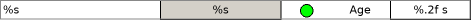
VISUALIZATION VISU_AlpacaGetBool  // 471x20
VAR_IN_OUT
	stInstance : ST_AlpacaGetBool;
END_VAR
    Rectangle (160,0 121x20), "%s", text variable: stInstance.bValue, colour toggle: stInstance.bValue
    Ellipse (300,4 13x13), colour toggle: stInstance.eStatusCode <> E_AlpacaStatusCode.OK
    Rectangle (0,0 161x20), "%s", text variable: stInstance.sName
    Rectangle (390,0 81x20), "%.2f s", text variable: stInstance.rAge
    Label (340,0 41x20), "Age"
END_VISUALIZATION

// ---- VISUs/Alpaca/VISU_AlpacaGetCoverState.TcVIS
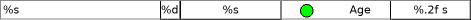
VISUALIZATION VISU_AlpacaGetCoverState  // 471x20
VAR_IN_OUT
	stInstance : ST_AlpacaGetCoverState;
END_VAR
    Rectangle (160,0 20x20), "%d", text variable: stInstance.nValue
    Rectangle (0,0 161x20), "%s", text variable: stInstance.sName
    Ellipse (300,4 13x13), colour toggle: stInstance.eStatusCode <> E_AlpacaStatusCode.OK
    Rectangle (390,0 81x20), "%.2f s", text variable: stInstance.rAge
    Label (340,0 41x20), "Age"
    Rectangle (180,0 101x20), "%s", text variable: stInstance.sValue
END_VISUALIZATION

// ---- VISUs/Alpaca/VISU_AlpacaGetLreal.TcVIS
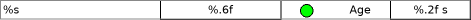
VISUALIZATION VISU_AlpacaGetLreal  // 471x20
VAR_IN_OUT
	stInstance : ST_AlpacaGetLreal;
END_VAR
    Rectangle (160,0 121x20), "%.6f", text variable: stInstance.lrValue
    Rectangle (0,0 161x20), "%s", text variable: stInstance.sName
    Ellipse (300,4 13x13), colour toggle: stInstance.eStatusCode <> E_AlpacaStatusCode.OK
    Rectangle (390,0 81x20), "%.2f s", text variable: stInstance.rAge
    Label (340,0 41x20), "Age"
END_VISUALIZATION

// ---- VISUs/Alpaca/VISU_AlpacaPutMove.TcVIS
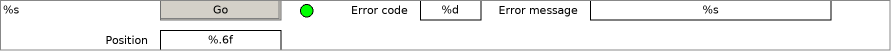
VISUALIZATION VISU_AlpacaPutMove  // 891x51
VAR_IN_OUT
	stInstance : ST_AlpacaPutMove;
END_VAR
    Frame (0,0 891x20)
        shows VISU_AlpacaPutRequest(stInstance := stInstance)
    Label (50,30 101x21), "Position"
    Rectangle (160,30 121x20), "%.6f", text variable: stInstance.i_Position
        OnMouseClick: write the text variable via Default
END_VISUALIZATION

// ---- VISUs/Alpaca/VISU_AlpacaPutNoArgs.TcVIS
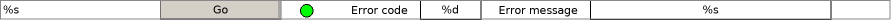
VISUALIZATION VISU_AlpacaPutNoArgs  // 891x20
VAR_IN_OUT
	stInstance : ST_AlpacaPutRequest;
END_VAR
    Frame (0,0 891x20)
        shows VISU_AlpacaPutRequest(stInstance := stInstance)
END_VISUALIZATION

// ---- VISUs/Alpaca/VISU_AlpacaPutRequest.TcVIS
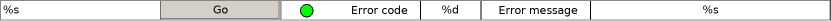
VISUALIZATION VISU_AlpacaPutRequest  // 831x21
VAR_IN_OUT
	stInstance : ST_AlpacaPutRequest;
END_VAR
    Rectangle (0,0 161x20), "%s", text variable: stInstance.sName
    Ellipse (300,4 13x13), colour toggle: stInstance.eStatusCode <> E_AlpacaStatusCode.OK
        p4168582468: stInstance.eStatusCode
    Button (160,0 121x20), "Go"
        OnMouseClick: execute { stInstance.bExecute := TRUE; }
    Label (350,0 61x21), "Error code"
    Rectangle (420,0 61x20), "%d", text variable: stInstance.nErrorCode
    Rectangle (590,0 241x20), "%s", text variable: stInstance.sErrorMessage
        p4168582468: stInstance.sErrorMessage
    Label (490,0 91x21), "Error message"
END_VISUALIZATION

// ---- VISUs/Alpaca/VISU_AlpacaPutSlewToAltAz.TcVIS
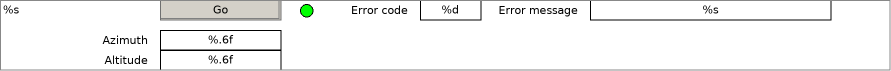
VISUALIZATION VISU_AlpacaPutSlewToAltAz  // 891x71
VAR_IN_OUT
	stInstance : ST_AlpacaPutSlewToAltAz;
END_VAR
    Frame (0,0 891x20)
        shows VISU_AlpacaPutRequest(stInstance := stInstance)
    Label (50,30 101x21), "Azimuth"
    Rectangle (160,30 121x20), "%.6f", text variable: stInstance.i_lrAzimuth
        OnMouseClick: write the text variable via Default
    Label (50,50 101x21), "Altitude"
    Rectangle (160,50 121x20), "%.6f", text variable: stInstance.i_lrAltitude
        OnMouseClick: write the text variable via Default
END_VISUALIZATION

// ---- VISUs/Alpaca/VISU_AlpacaPutSlewToCoordinates.TcVIS
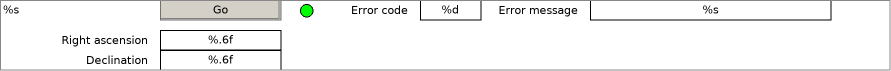
VISUALIZATION VISU_AlpacaPutSlewToCoordinates  // 891x71
VAR_IN_OUT
	stInstance : ST_AlpacaPutSlewToCoordinates;
END_VAR
    Frame (0,0 891x20)
        shows VISU_AlpacaPutRequest(stInstance := stInstance)
    Label (50,30 101x21), "Right ascension"
    Rectangle (160,30 121x20), "%.6f", text variable: stInstance.i_lrRightAscension
        OnMouseClick: write the text variable via Default
    Label (50,50 101x21), "Declination"
    Rectangle (160,50 121x20), "%.6f", text variable: stInstance.i_lrDeclination
        OnMouseClick: write the text variable via Default
END_VISUALIZATION

// ---- VISUs/Alpaca/VISU_AlpacaPutTracking.TcVIS
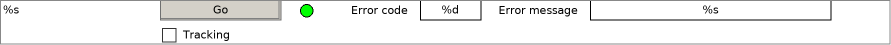
VISUALIZATION VISU_AlpacaPutTracking  // 891x45
VAR_IN_OUT
	stInstance : ST_AlpacaPutTracking;
END_VAR
    Frame (0,0 891x20)
        shows VISU_AlpacaPutRequest(stInstance := stInstance)
    Checkbox (160,25 121x20), "Tracking", variable: stInstance.i_bTracking
END_VISUALIZATION

// ---- VISUs/AsaTelescope/VISU_AsaTelescope.TcVIS
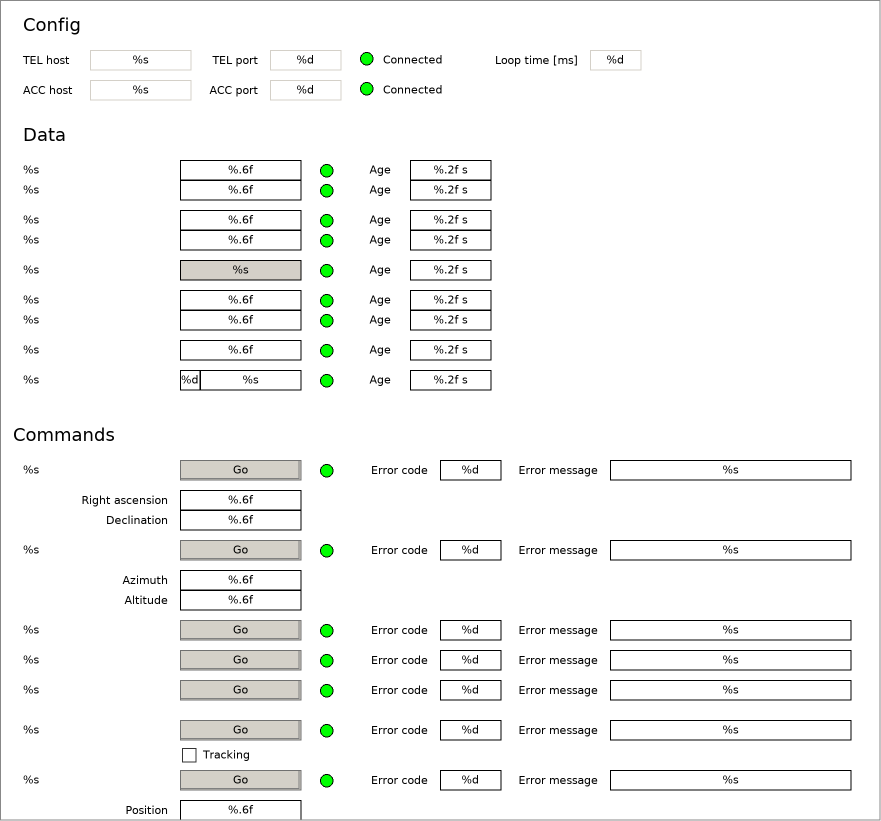
VISUALIZATION VISU_AsaTelescope  // 881x821
VAR_IN_OUT
	fbInstance : FB_AsaTelescope;
END_VAR
    Frame (20,160 511x20)
        shows VISU_AlpacaGetLreal(stInstance := fbInstance.stData.stRightAscension)
    Frame (20,180 511x20)
        shows VISU_AlpacaGetLreal(stInstance := fbInstance.stData.stDeclination)
    Frame (20,210 511x20)
        shows VISU_AlpacaGetLreal(stInstance := fbInstance.stData.stAzimuth)
    Frame (20,230 511x20)
        shows VISU_AlpacaGetLreal(stInstance := fbInstance.stData.stAltitude)
    Frame (20,290 511x20)
        shows VISU_AlpacaGetLreal(stInstance := fbInstance.stData.stTargetRightAscension)
    Frame (20,310 511x20)
        shows VISU_AlpacaGetLreal(stInstance := fbInstance.stData.stTargetDeclination)
    Frame (20,260 511x20)
        shows VISU_AlpacaGetBool(stInstance := fbInstance.stData.stSlewing)
    Label (20,120 150x30), "Data"
    Label (10,420 211x30), "Commands"
    Frame (20,460 861x81)
        shows VISU_AlpacaPutSlewToCoordinates(stInstance := fbInstance.stCommands.stSlewToCoo)
    Frame (20,540 861x81)
        shows VISU_AlpacaPutSlewToAltAz(stInstance := fbInstance.stCommands.stSlewToAltAz)
    Frame (20,650 861x20)
        shows VISU_AlpacaPutNoArgs(stInstance := fbInstance.stCommands.stOpenCover)
    Frame (20,680 861x20)
        shows VISU_AlpacaPutNoArgs(stInstance := fbInstance.stCommands.stCloseCover)
    Frame (20,720 861x51)
        shows VISU_AlpacaPutTracking(stInstance := fbInstance.stCommands.stTracking)
    Frame (20,340 511x20)
        shows VISU_AlpacaGetLreal(stInstance := fbInstance.stData.stM2Position)
    Frame (20,770 861x51)
        shows VISU_AlpacaPutMove(stInstance := fbInstance.stCommands.stM2Move)
    Frame (20,370 511x20)
        shows VISU_AlpacaGetCoverState(stInstance := fbInstance.stData.stCoverState)
    Frame (20,620 861x20)
        shows VISU_AlpacaPutNoArgs(stInstance := fbInstance.stCommands.stAbortSlew)
    Label (20,10 150x30), "Config"
    Label (20,50 71x21), "TEL host"
    Textfield (90,50 101x20), "%s", text variable: fbInstance.sTelHost
        OnMouseClick: write the text variable via Default
    Textfield (270,50 71x20), "%d", text variable: fbInstance.nTelPort
        OnMouseClick: write the text variable via Default
    Label (200,50 61x21), "TEL port"
    Textfield (590,50 51x20), "%d", text variable: fbInstance.nLoopTime
        OnMouseClick: write the text variable via Default
    Label (490,50 91x21), "Loop time [ms]"
    Label (20,80 71x21), "ACC host"
    Textfield (90,80 101x20), "%s", text variable: fbInstance.sAccHost
        OnMouseClick: write the text variable via Default
    Textfield (270,80 71x20), "%d", text variable: fbInstance.nAccPort
        OnMouseClick: write the text variable via Default
    Label (200,80 61x21), "ACC port"
    Ellipse (360,52 13x13), colour toggle: NOT fbInstance.bTelConnected
    Ellipse (360,82 13x13), colour toggle: NOT fbInstance.bAccConnected
    Label (380,50 91x20), "Connected"
    Label (380,80 91x20), "Connected"
END_VISUALIZATION

// ---- VISUs/VISU_MAIN.TcVIS
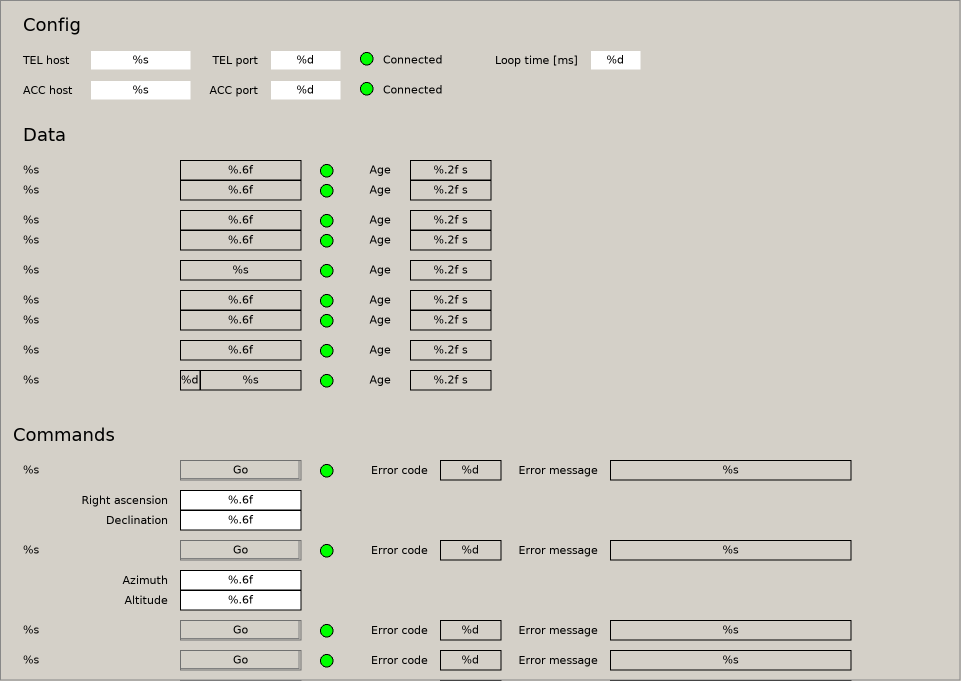
VISUALIZATION VISU_MAIN  // 961x681
    Frame (0,0 961x681)
        shows VISU_AsaTelescope(fbInstance := MAIN.fbTelescope)
END_VISUALIZATION
